PROGRAM MAIN
VAR
END_VAR

END_PROGRAM

(* stored: Version 1.1.0.1
   POU MAIN: Id {272197ff-b391-4f07-8aec-ea8e94a0d1dd} *)
